// TIA Portal V17 export
// export: Created 2025-03-05T08:03:01.0643291Z, ExportSetting WithDefaults, DisplayName Totally Integrated Automation Portal, DisplayVersion V17 Update 8, DisplayName TIA Portal Openness, DisplayVersion V17 Update 8, DisplayName TIA Portal Version Control Interface, DisplayVersion V17, DisplayName SINAMICS Startdrive Advanced, DisplayVersion V17 SP2, DisplayName SINAMICS Startdrive G110M, G120, G120C, G120D, G120P, G115D, DisplayVersion V17 SP2, DisplayName SINAMICS Startdrive G130, G150, S120, S150, SINAMICS MV, S210, DisplayVersion V17 SP2, DisplayName STEP 7 Professional, DisplayVersion V17 Update 8, DisplayName SINUMERIK ONE STEP 7 Toolbox, DisplayVersion V17 Update 12, DisplayName SINUMERIK 840D sl STEP 7 Toolbox, DisplayVersion V17 Update 12, DisplayName STEP 7 Safety, DisplayVersion V17 Update 6, DisplayName WinCC Advanced, DisplayVersion V17 Update 8
DATA_BLOCK "DB16727_POWDER_FLOW_DATA_SAVE_U02_COMBINER"   // DB16727
{ DB_Accessible_From_OPC_UA := 'FALSE' }
VERSION : 0.1
// stored: AutoNumber false, DBAccessibleFromOPCUA false, DBAccessibleFromWebserver true, InstanceOfName FB16700_POWDER_FLOW_DATA_SAVE, InstanceOfType FB
"FB16700_POWDER_FLOW_DATA_SAVE"
   // VAR_INPUT
   //    iMEDICOAT_DATA : Int;
   // END_VAR
   // VAR_OUTPUT
   //    oMEDICOAT_DATA_ARRAY : Array[1..20] of "MEDICOAT_TIME_STAMP";
   // END_VAR
   // VAR_IN_OUT
   //    ARRAY_NUMBER_MEMORY : Int;
   // END_VAR
   // VAR
   //    SAVE_VALUE_TRIGGER_TON : TON_TIME;
   //    RESET_VALUE_TON { S7_SetPoint := 'True'} : TON_TIME;
   //    SAVE_VALUE_TRIGGER { S7_SetPoint := 'True'} : Bool;
   //    RESET_TIMER_AUX : Bool;
   //    PULSE_AUX : Bool;
   // END_VAR
BEGIN
END_DATA_BLOCK
